FUNCTION_BLOCK HandShakeMech_Rec (* Basic Function Block Type *)
  (* Standard: 61499-2 *)
  (* Version 0.0, 11/3/2020, prana, nxtControl GmbH, Template *)
  PACKAGE Main;
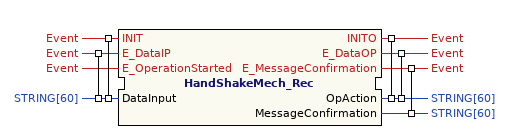
  EVENT_INPUT
    INIT WITH DataInput; (* Initialization Request *)
    E_DataIP WITH DataInput; (* Normal Execution Request *)
    E_OperationStarted;
  END_EVENT
  EVENT_OUTPUT
    INITO WITH OpAction; (* Initialization Confirm *)
    E_DataOP WITH OpAction; (* Execution Confirmation *)
    E_MessageConfirmation WITH MessageConfirmation;
  END_EVENT
  VAR_INPUT
    DataInput : STRING[60]; (* Input event qualifier *)
  END_VAR
  VAR_OUTPUT
    OpAction : STRING[60]; (* Output event qualifier *)
    MessageConfirmation : STRING[60];
  END_VAR
  VAR
    i : INT;
    j : INT;
    l : INT;
    c : INT;
    prevCount : STRING[60];
    prevCommand : STRING[60] := '';
    OperationStarted : BOOL := FALSE;
    CurrentCommand : STRING[60];
    CurrentCount : STRING[60];
    ResendConfirmation : BOOL;
    RestartOperation : BOOL;
    StartOperation : BOOL;
  END_VAR
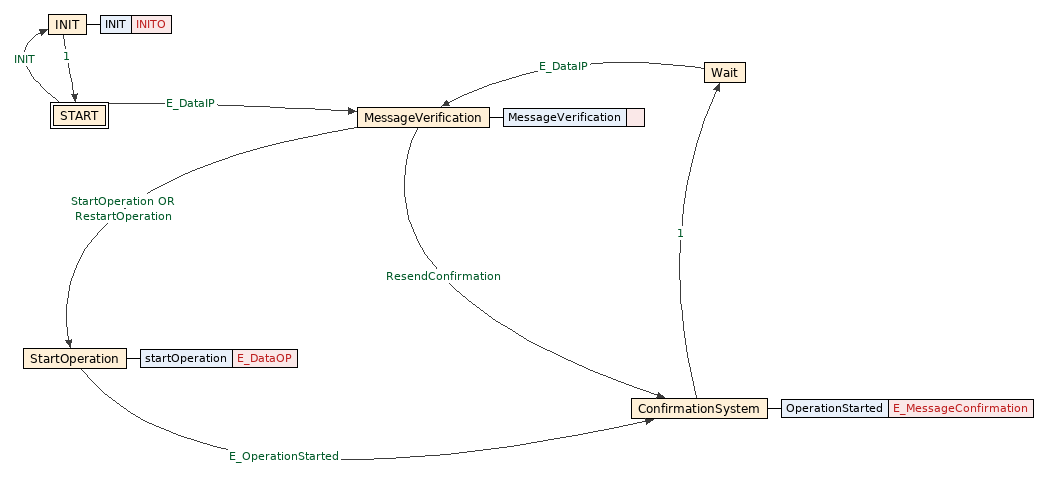
  EC_STATES
    START; (* Initial State *)
    INIT : INIT -> INITO; (* Initialization *)
    MessageVerification : MessageVerification;
    ConfirmationSystem : OperationStarted -> E_MessageConfirmation;
    Wait;
    StartOperation : startOperation -> E_DataOP;
  END_STATES
  EC_TRANSITIONS
    START TO INIT := INIT;
    INIT TO START := 1;
    START TO MessageVerification := E_DataIP;
    ConfirmationSystem TO Wait := 1;
    Wait TO MessageVerification := E_DataIP;
    MessageVerification TO StartOperation := StartOperation OR RestartOperation;
    StartOperation TO ConfirmationSystem := E_OperationStarted;
    MessageVerification TO ConfirmationSystem := ResendConfirmation;
  END_TRANSITIONS
  ALGORITHM INIT IN ST: (* Initialization algorithm *)
prevCommand := '';
OperationStarted := FALSE;
  END_ALGORITHM
  ALGORITHM MessageVerification IN ST:
// Datainput example: C2_to_C5,2


i := DINT_TO_INT(FIND(DataInput,':'));
i := i - 1;
CurrentCommand := LEFT(DataInput,i);  //seperate message count from action information eg: C2_to_C5

l := DINT_TO_INT(LEN(DataInput));
c := l - (DINT_TO_INT(FIND(DataInput,':')));
CurrentCount := RIGHT(DataInput,c);    //Store Message count.... eg: 2 from above example


IF CurrentCount = '1' THEN
	StartOperation := TRUE;

ELSIF CurrentCount <> '1' THEN
	IF (CurrentCommand = prevCommand) & (OperationStarted) THEN
		ResendConfirmation := TRUE;
	ELSIF (CurrentCommand = prevCommand) & (NOT OperationStarted) THEN
		RestartOperation := TRUE;
	ELSIF (CurrentCommand <> prevCommand) THEN
		StartOperation := TRUE;
	END_IF;
END_IF;

prevCommand := CurrentCommand;
prevCount := CurrentCount;
OperationStarted := FALSE;
  END_ALGORITHM
  ALGORITHM OperationStarted IN ST:
MessageConfirmation := CONCAT(DataInput,';R');
ResendConfirmation := FALSE;
OperationStarted := TRUE;
  END_ALGORITHM
  ALGORITHM startOperation IN ST:
OpAction := CurrentCommand;

RestartOperation := FALSE;
StartOperation := FALSE;
  END_ALGORITHM
END_FUNCTION_BLOCK
